// Mitsubishi GX Works2 project: BookEX6_50 Positionning   PLC: Q13UDV

// global labels: Global
VAR_GLOBAL
  bVar0 AT M5000 : BOOL;
  abArray0 AT M5010 : ARRAY [0..49] OF BOOL;
  sStr0 AT D5000 : STRING[199];
  sStr1 AT D5100 : STRING[199];
  sStr2 AT D5200 : STRING[199];
  sStr3 AT D5300 : STRING[199];
  sStr4 AT D5400 : STRING[199];
  sStr5 AT D5500 : STRING[199];
  sStr6 AT D5600 : STRING[199];
  sStr7 AT D5700 : STRING[199];
  sStr8 AT D5800 : STRING[199];
  sStr9 AT D5900 : STRING[199];
  iVar0 AT D4500 : INT;
  iVar1 AT D4501 : INT;
  iVar2 AT D4502 : INT;
  iVar3 AT D4503 : INT;
  iVar4 AT D4504 : INT;
  iVar5 AT D4505 : INT;
  iVar6 AT D4506 : INT;
  iVar7 AT D4507 : INT;
  iVar8 AT D4508 : INT;
  iVar9 AT D4509 : INT;
  dVar0 AT D4510 : DINT;
  dVar1 AT D4512 : DINT;
  dVar2 AT D4514 : DINT;
  dVar3 AT D4516 : DINT;
  dVar4 AT D4518 : DINT;
  dVar5 AT D4520 : DINT;
  dVar6 AT D4522 : DINT;
  dVar7 AT D4524 : DINT;
  dVar8 AT D4526 : DINT;
  dVar9 AT D4528 : DINT;
  wVar0 AT D4530 : WORD;
  wVar1 AT D4531 : WORD;
  wVar2 AT D4532 : WORD;
  wVar3 AT D4533 : WORD;
  wVar4 AT D4534 : WORD;
  wVar5 AT D4535 : WORD;
  wVar6 AT D4536 : WORD;
  wVar7 AT D4537 : WORD;
  wVar8 AT D4538 : WORD;
  wVar9 AT D4539 : WORD;
  dwVar0 AT D4540 : DWORD;
  dwVar1 AT D4542 : DWORD;
  dwVar2 AT D4544 : DWORD;
  dwVar3 AT D4546 : DWORD;
  dwVar4 AT D4548 : DWORD;
  dwVar5 AT D4550 : DWORD;
  dwVar6 AT D4552 : DWORD;
  dwVar7 AT D4554 : DWORD;
  dwVar8 AT D4556 : DWORD;
  dwVar9 AT D4558 : DWORD;
  fsVar0 AT D4560 : REAL;
  fsVar1 AT D4562 : REAL;
  fsVar2 AT D4564 : REAL;
  fsVar3 AT D4566 : REAL;
  fsVar4 AT D4568 : REAL;
  fsVar5 AT D4570 : REAL;
  fsVar6 AT D4572 : REAL;
  fsVar7 AT D4574 : REAL;
  fsVar8 AT D4576 : REAL;
  fsVar9 AT D4578 : REAL;
  fdVar0 AT D4580 : LREAL;
  tTime0 AT D4620 : TIME;
  tTime1 AT D4622 : TIME;
  tTime2 AT D4624 : TIME;
  tTime3 AT D4626 : TIME;
  tTime4 AT D4628 : TIME;
  tTime5 AT D4630 : TIME;
  tTime6 AT D4632 : TIME;
  tTime7 AT D4634 : TIME;
  tTime8 AT D4636 : TIME;
  tTime9 AT D4638 : TIME;
  tTime10 AT D4640 : TIME;
  bVar1 AT M5001 : BOOL;
  bVar2 AT M5002 : BOOL;
  bVar3 AT M5003 : BOOL;
  bVar4 AT M5004 : BOOL;
  bVar5 AT M5005 : BOOL;
  bVar6 AT M5006 : BOOL;
  bVar7 AT M5007 : BOOL;
  bVar8 AT M5008 : BOOL;
  bVar9 AT M5009 : BOOL;
  abArray1 AT M5060 : ARRAY [0..49] OF BOOL;
  abArray2 AT M5110 : ARRAY [0..49] OF BOOL;
  abArray3 AT M5160 : ARRAY [0..49] OF BOOL;
  abArray4 AT M5210 : ARRAY [0..49] OF BOOL;
  abArray5 AT M5260 : ARRAY [0..49] OF BOOL;
  abArray6 AT M5310 : ARRAY [0..49] OF BOOL;
  abArray7 AT M5360 : ARRAY [0..49] OF BOOL;
  abArray8 AT M5410 : ARRAY [0..49] OF BOOL;
  abArray9 AT M5460 : ARRAY [0..49] OF BOOL;
  fdVar1 AT D4584 : LREAL;
  fdVar2 AT D4588 : LREAL;
  fdVar3 AT D4592 : LREAL;
  fdVar4 AT D4596 : LREAL;
  fdVar5 AT D4600 : LREAL;
  fdVar6 AT D4604 : LREAL;
  fdVar7 AT D4608 : LREAL;
  fdVar8 AT D4612 : LREAL;
  fdVar9 AT D4616 : LREAL;
  afsPen0 AT D2000 : ARRAY [0..499] OF REAL;
  afsPen1 AT D3000 : ARRAY [0..499] OF REAL;
END_VAR
// user libraries (not included): HMI

PROGRAM ExPINIT
VAR
  bReqCmd : BOOL;
  bExeFlag : BOOL;
  bMemFlag : BOOL;
  aCtrlData : ARRAY [0..1] OF INT;
  abComp : ARRAY [0..1] OF BOOL;
  iErrCode : INT;
END_VAR
(* structured ladder/FBD written out as ST: instructions are called as NAME(EN, inputs, outputs); _pN, _eN, _tN stand for wires *)
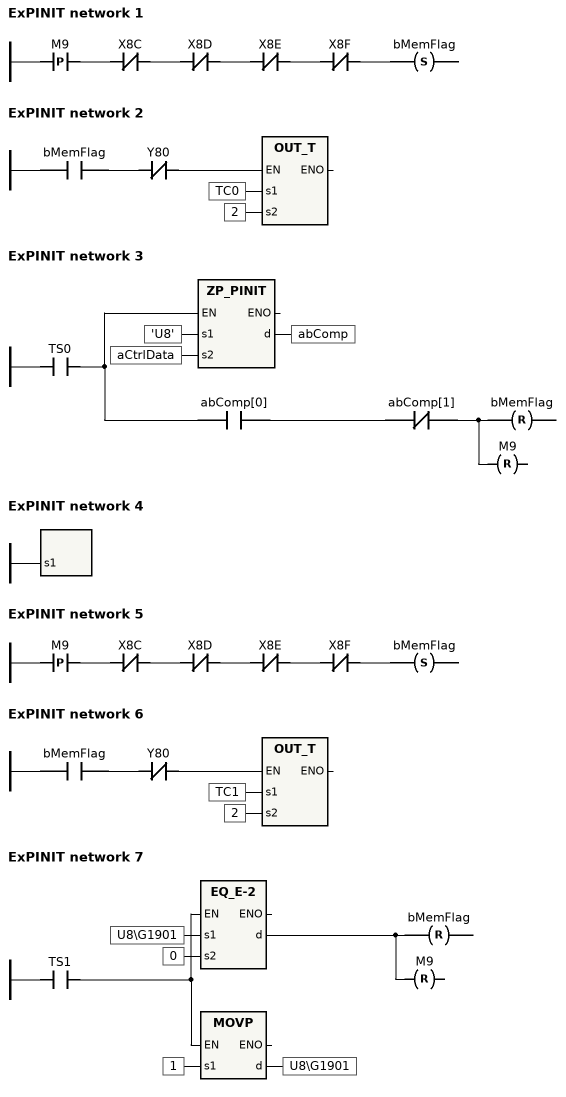
(* network 1 *)
SET(LDP(TRUE, M9) AND NOT X8C AND NOT X8D AND NOT X8E AND NOT X8F, bMemFlag);
(* network 2 *)
OUT_T(bMemFlag AND NOT Y80, TC0, 2);
(* network 3 *)
ZP_PINIT(TS0, 'U8', aCtrlData, abComp);
_p1 := TS0 AND abComp[0] AND NOT abComp[1];
RST(_p1, bMemFlag);
RST(_p1, M9);
(* network 4 *)
(* element kind 10  <- TRUE *)
(* network 5 *)
SET(LDP(TRUE, M9) AND NOT X8C AND NOT X8D AND NOT X8E AND NOT X8F, bMemFlag);
(* network 6 *)
OUT_T(bMemFlag AND NOT Y80, TC1, 2);
(* network 7 *)
MOVP(TS1, 1, U8\G1901);
EQ_E(TS1, U8\G1901, 0, _t1);
RST(_t1, bMemFlag);
RST(_t1, M9);
END_PROGRAM

PROGRAM ExABRST
VAR
  bReqCmd : BOOL;
  bExeFlag : BOOL;
  bMemFlag : BOOL;
  aCtrlData : ARRAY [0..7] OF INT;
  abComp : ARRAY [0..1] OF BOOL;
  iErrCode : INT;
END_VAR
(* structured ladder/FBD written out as ST: instructions are called as NAME(EN, inputs, outputs); _pN, _eN, _tN stand for wires *)
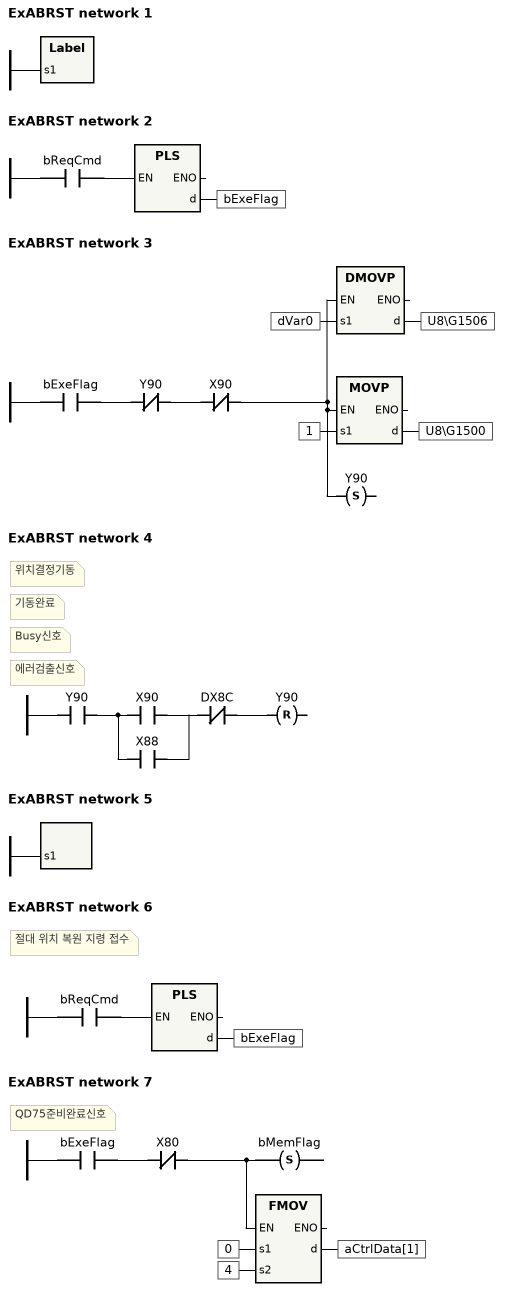
(* network 1 *)
(* element kind 9 Label <- TRUE *)
(* network 2 *)
PLS(bReqCmd, bExeFlag);
(* network 3 *)
_p1 := bExeFlag AND NOT Y90 AND NOT X90;
DMOVP(_p1, dVar0, U8\G1506);
MOVP(_p1, 1, U8\G1500);
SET(_p1, Y90);
(* network 4 *)
(* 위치결정기동 *)
(* 기동완료 *)
(* Busy신호 *)
(* 에러검출신호 *)
RST(((Y90 AND X90) OR (Y90 AND X88)) AND NOT DX8C, Y90);
(* network 5 *)
(* element kind 10  <- TRUE *)
(* network 6 Label: *)
(* 절대 위치 복원 지령 접수 *)
PLS(bReqCmd, bExeFlag);
(* network 7 *)
(* QD75준비완료신호 *)
_p1 := bExeFlag AND NOT X80;
SET(_p1, bMemFlag);
FMOV(_p1, 0, 4, aCtrlData[1]);
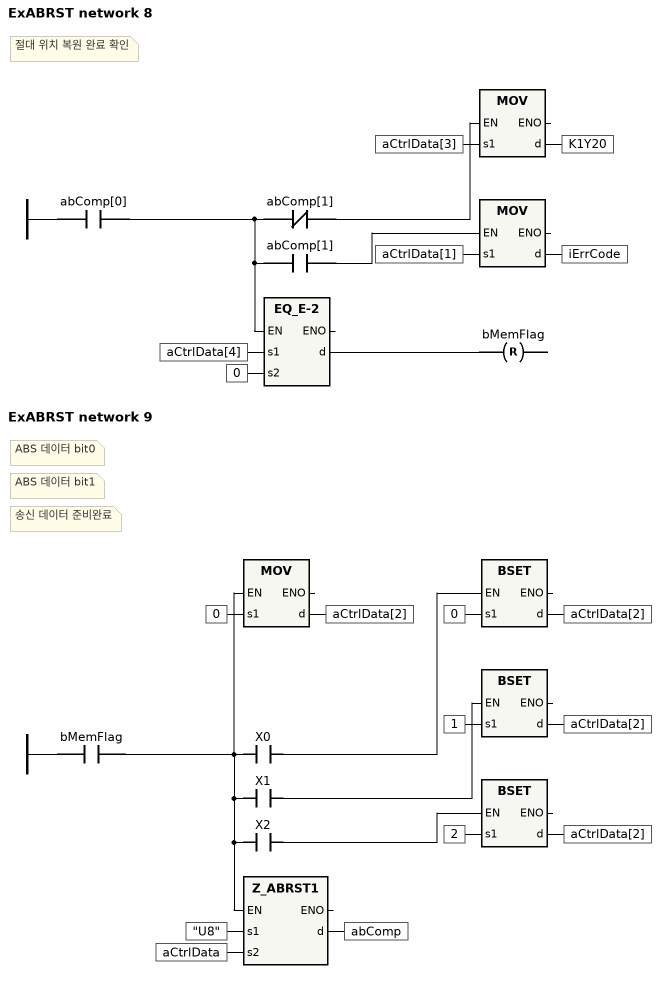
(* network 8 *)
(* 절대 위치 복원 완료 확인 *)
MOV(abComp[0] AND NOT abComp[1], aCtrlData[3], K1Y20);
MOV(abComp[0] AND abComp[1], aCtrlData[1], iErrCode);
EQ_E(abComp[0], aCtrlData[4], 0, _t1);
RST(_t1, bMemFlag);
(* network 9 *)
(* ABS 데이터 bit0 *)
(* ABS 데이터 bit1 *)
(* 송신 데이터 준비완료 *)
MOV(bMemFlag, 0, aCtrlData[2]);
BSET(bMemFlag AND X0, 0, aCtrlData[2]);
BSET(bMemFlag AND X1, 1, aCtrlData[2]);
BSET(bMemFlag AND X2, 2, aCtrlData[2]);
Z_ABRST1(bMemFlag, "U8", aCtrlData, abComp);
END_PROGRAM

PROGRAM ExPSTRT
VAR
  bReqCmd : BOOL;
  bExeFlag : BOOL;
  bMemFlag : BOOL;
  aCtrlData : ARRAY [0..2] OF INT;
  abComp : ARRAY [0..1] OF BOOL;
  iErrCode : INT;
END_VAR
(* structured ladder/FBD written out as ST: instructions are called as NAME(EN, inputs, outputs); _pN, _eN, _tN stand for wires *)
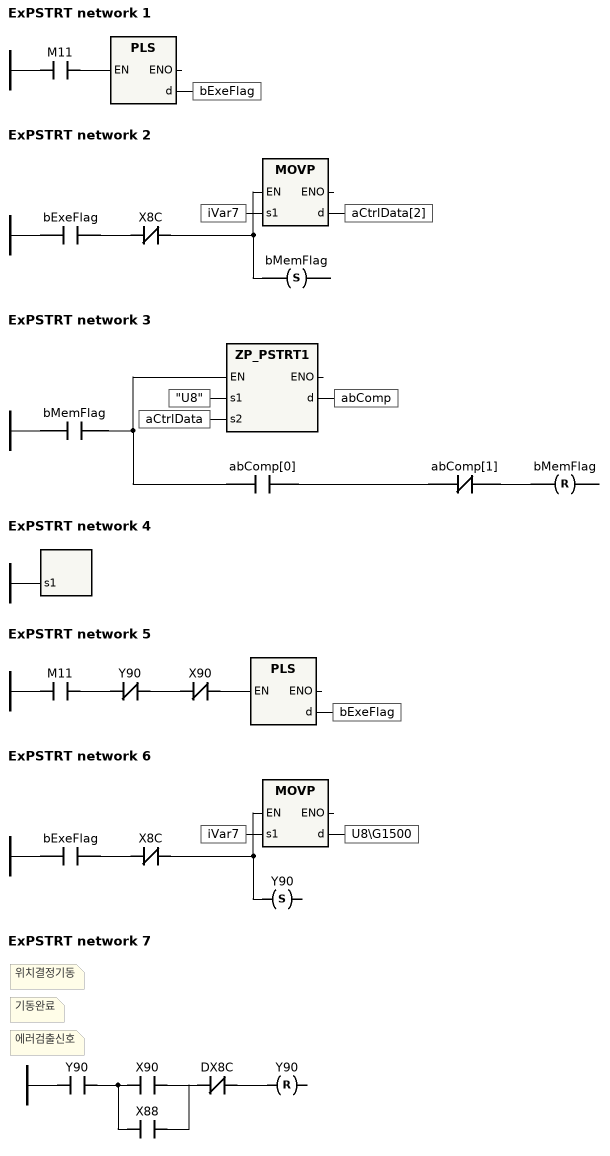
(* network 1 *)
PLS(M11, bExeFlag);
(* network 2 *)
_p1 := bExeFlag AND NOT X8C;
MOVP(_p1, iVar7, aCtrlData[2]);
SET(_p1, bMemFlag);
(* network 3 *)
ZP_PSTRT1(bMemFlag, "U8", aCtrlData, abComp);
RST(bMemFlag AND abComp[0] AND NOT abComp[1], bMemFlag);
(* network 4 *)
(* element kind 10  <- TRUE *)
(* network 5 Label: *)
PLS(M11 AND NOT Y90 AND NOT X90, bExeFlag);
(* network 6 *)
_p1 := bExeFlag AND NOT X8C;
MOVP(_p1, iVar7, U8\G1500);
SET(_p1, Y90);
(* network 7 *)
(* 위치결정기동 *)
(* 기동완료 *)
(* 에러검출신호 *)
RST(((Y90 AND X90) OR (Y90 AND X88)) AND NOT DX8C, Y90);
END_PROGRAM

PROGRAM ExTEACH
VAR
  bReqCmd : BOOL;
  bExeFlag : BOOL;
  bMemFlag : BOOL;
  aCtrlData : ARRAY [0..3] OF INT;
  abComp : ARRAY [0..1] OF BOOL;
  iErrCode : INT;
END_VAR
(* structured ladder/FBD written out as ST: instructions are called as NAME(EN, inputs, outputs); _pN, _eN, _tN stand for wires *)
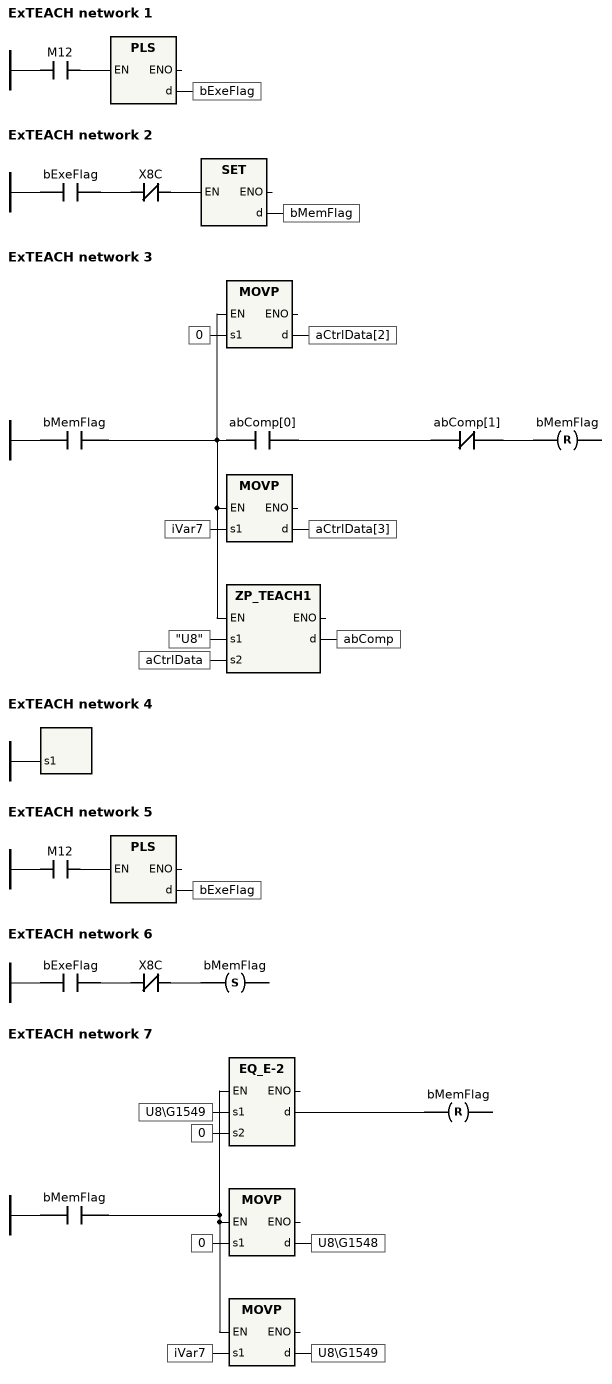
(* network 1 *)
PLS(M12, bExeFlag);
(* network 2 *)
SET(bExeFlag AND NOT X8C, bMemFlag);
(* network 3 *)
MOVP(bMemFlag, 0, aCtrlData[2]);
MOVP(bMemFlag, iVar7, aCtrlData[3]);
ZP_TEACH1(bMemFlag, "U8", aCtrlData, abComp);
RST(bMemFlag AND abComp[0] AND NOT abComp[1], bMemFlag);
(* network 4 *)
(* element kind 10  <- TRUE *)
(* network 5 *)
PLS(M12, bExeFlag);
(* network 6 *)
SET(bExeFlag AND NOT X8C, bMemFlag);
(* network 7 *)
MOVP(bMemFlag, 0, U8\G1548);
MOVP(bMemFlag, iVar7, U8\G1549);
EQ_E(bMemFlag, U8\G1549, 0, _t1);
RST(_t1, bMemFlag);
END_PROGRAM

PROGRAM ExPFWRT
VAR
  bReqCmd : BOOL;
  bExeFlag : BOOL;
  bMemFlag : BOOL;
  aCtrlData : ARRAY [0..1] OF INT;
  abComp : ARRAY [0..1] OF BOOL;
  iErrCode : INT;
END_VAR
(* structured ladder/FBD written out as ST: instructions are called as NAME(EN, inputs, outputs); _pN, _eN, _tN stand for wires *)
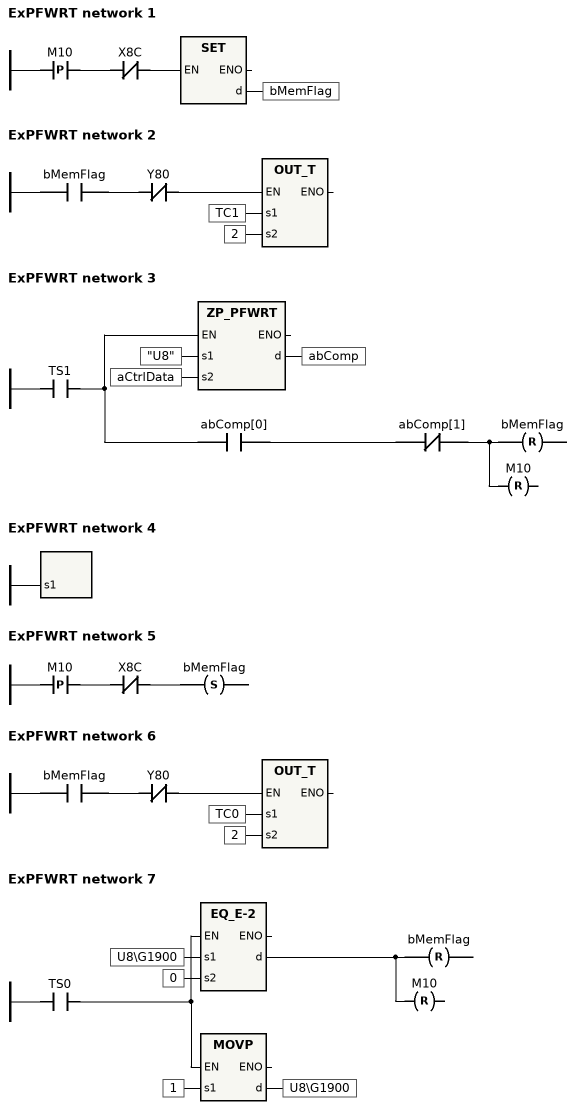
(* network 1 *)
SET(LDP(TRUE, M10) AND NOT X8C, bMemFlag);
(* network 2 *)
OUT_T(bMemFlag AND NOT Y80, TC1, 2);
(* network 3 *)
ZP_PFWRT(TS1, "U8", aCtrlData, abComp);
_p1 := TS1 AND abComp[0] AND NOT abComp[1];
RST(_p1, bMemFlag);
RST(_p1, M10);
(* network 4 *)
(* element kind 10  <- TRUE *)
(* network 5 *)
SET(LDP(TRUE, M10) AND NOT X8C, bMemFlag);
(* network 6 *)
OUT_T(bMemFlag AND NOT Y80, TC0, 2);
(* network 7 *)
MOVP(TS0, 1, U8\G1900);
EQ_E(TS0, U8\G1900, 0, _t1);
RST(_t1, bMemFlag);
RST(_t1, M10);
END_PROGRAM

FUNCTION_BLOCK ms2Ready
VAR_INPUT
  b_EN : BOOL;
  i_Start_IO_No : INT;  (* Module XY addr *)
END_VAR
VAR_OUTPUT
  b_ENO : BOOL;
  b_Ready : BOOL;
END_VAR
VAR
  bRdy77 : BOOL;
  bRdyCPU : BOOL;
END_VAR
VAR_OUTPUT
  b_AllAxis : BOOL;
  b_OK : BOOL;
END_VAR
VAR
  bSync77 : BOOL;
  bReady : BOOL;
  bAllAxis : BOOL;
END_VAR
;
b_ENO := b_EN;
Z0 := i_Start_IO_No * 16;
bRdy77 := X0Z0;
bSync77 := X1Z0;
bRdyCPU := Y0Z0;

IF NOT b_EN  THEN
	bReady := FALSE;
	bAllAxis := FALSE;
	b_OK := FALSE;
ELSE
	bReady := NOT SM0;
	bAllAxis := bRdyCPU AND bSync77;
	b_OK := bRdyCPU AND bRdy77 AND bSync77;
END_IF;

b_Ready := bReady;
b_AllAxis := bAllAxis;
END_FUNCTION_BLOCK

FUNCTION_BLOCK ms2Status
VAR_INPUT
  b_EN : BOOL;
  i_Start_IO_No : INT;  (* Module XY addr *)
  i_Axis : INT;  (* Axis No *)
END_VAR
VAR_OUTPUT
  b_ENO : BOOL;
  i_Status : INT;
  i_Error : INT;
END_VAR
VAR
  bRes : BOOL;
  AxisOff : INT;
  iTmp : INT;
END_VAR
VAR_OUTPUT
  d_CurrVal : DINT;
END_VAR
VAR
  dTmp : DINT;
END_VAR
VAR_OUTPUT
  d_CurrSpd : DINT;
  i_Warn : INT;
  d_TargVal : DINT;
  d_TargSpd : DINT;
  d_MacVal : DINT;
  w_Flag : WORD;
  w_Signal : WORD;
END_VAR
;
b_ENO := b_EN;
IF NOT LDP(TRUE, b_EN) THEN
	RETURN;
END_IF;
AxisOff := (i_Axis - 1) * 100;
bRes := FROM( TRUE, i_Start_IO_No, AxisOff+809, 1, iTmp);
i_Status := iTmp;
bRes := FROM( TRUE, i_Start_IO_No, AxisOff+806, 1, iTmp);
i_Error := iTmp;
bRes := FROM( TRUE, i_Start_IO_No, AxisOff+807, 1, iTmp);
i_Warn := iTmp;
bRes := DFRO( TRUE, i_Start_IO_No, AxisOff+800, 1, dTmp);
d_CurrVal := dTmp;
bRes := DFRO( TRUE, i_Start_IO_No, AxisOff+802, 1, dTmp);
d_MacVal := dTmp;
bRes := DFRO( TRUE, i_Start_IO_No, AxisOff+810, 1, dTmp);
d_CurrSpd := dTmp;
bRes := DFRO( TRUE, i_Start_IO_No, AxisOff+818, 1, dTmp);
d_TargVal := dTmp;
bRes := DFRO( TRUE, i_Start_IO_No, AxisOff+820, 1, dTmp);
d_TargSpd := dTmp;
bRes := FROM( TRUE, i_Start_IO_No, AxisOff+817, 1, iTmp);
w_Flag := INT_TO_WORD(iTmp);
bRes := FROM( TRUE, i_Start_IO_No, AxisOff+816, 1, iTmp);
w_Signal := INT_TO_WORD(iTmp);

(* 축 동작상태
		-2：스텝 대기중
		-1：에러 발생중
		0：대기중
		1：정지중
		2：보간중
		3：JOG 운전중
		4：수동 펄서 운전중
		5：해석중
		6：특수 기동 대기중
		7：원점복귀중
		8：위치제어중
		9：속도제어중
		10：속도·위치제어의 속도제어중
		11：속도·위치제어의 위치제어중
		12：위치·속도제어의 위치제어중
		13：위치·속도제어의 속도제어중
		15：동기제어중
		20：서보 미접속/서보앰프 전원 OFF
		21：서보 OFF 중
		30：제어모드 전환중
		31：속도 제어 모드중
		32：토크 제어 모드중
		33：스톱퍼 제어 모드중
*)
END_FUNCTION_BLOCK

FUNCTION_BLOCK ms2JOG
VAR_INPUT
  b_EN : BOOL;
  i_Start_IO_No : INT;  (* Module XY addr *)
  i_Axis : INT;  (* Axis No *)
  b_CW : BOOL;
  b_CCW : BOOL;
  d_JOGSpd : DINT;
END_VAR
VAR_OUTPUT
  b_ENO : BOOL;
END_VAR
VAR
  bRes : BOOL;
  AxisOff : INT;
  bError : BOOL;
  bBusy : BOOL;
  bReady : BOOL;
  bCW : BOOL;
  bCCW : BOOL;
END_VAR
VAR_INPUT
  b_SetSp : BOOL;
END_VAR
VAR
  bRun : BOOL;
  iCmd : INT;
END_VAR
;
b_ENO := b_EN;
Z0 := i_Start_IO_No * 16;
Z1 := Z0 + i_Axis - 1;
AxisOff := (i_Axis - 1) * 100;
bReady := X0Z0;
bError := X8Z1;
bBusy := XCZ0;

IF LDP(TRUE, b_SetSp) THEN
	bRes	:= TO( TRUE, 0, i_Start_IO_No, AxisOff+1517, 1);
	bRes	:= DTO( TRUE, d_JOGSpd * 10000, i_Start_IO_No, AxisOff+1518, 1);
END_IF;
iCmd := BOOL_TO_INT(b_CW) + BOOL_TO_INT(b_CCW) * 2;
CASE iCmd OF
	0, 3 : 	bCW := FALSE;
				bCCW := FALSE;
	1 : (* CW *)
				bCW := 	bReady AND NOT bError;
	2 : (* CCW *)
				bCCW := 	bReady AND NOT bError;
END_CASE;			 

Y8Z0 :=	bCCW;
Y9Z0 := bCW;
END_FUNCTION_BLOCK

PROGRAM ExJOG
VAR
  RunJog : BOOL;
  ServoRdy : BOOL;
  ReqHOFF : BOOL;
  MemHOFF : BOOL;
  wTmp : WORD;
  CmdHOFF : BOOL;
  ReqHPR : BOOL;
  ReqStop : BOOL;
END_VAR
(* structured ladder/FBD written out as ST: instructions are called as NAME(EN, inputs, outputs); _pN, _eN, _tN stand for wires *)
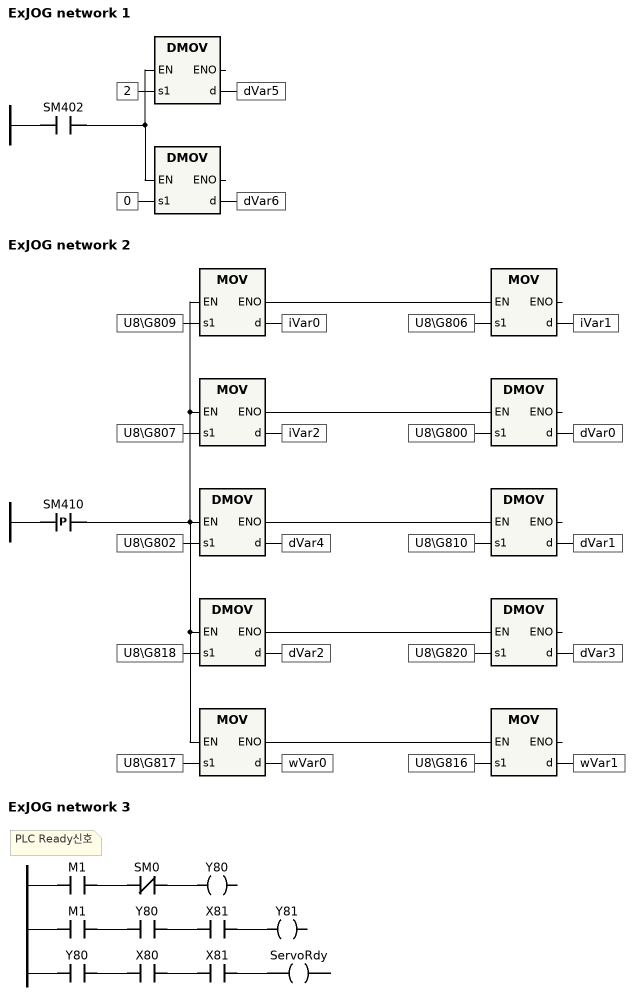
(* network 1 *)
DMOV(SM402, 2, dVar5);
DMOV(SM402, 0, dVar6);
(* network 2 *)
_p1 := LDP(TRUE, SM410);
_e2 := MOV(_p1, U8\G809, iVar0);
MOV(_e2, U8\G806, iVar1);
_e3 := MOV(_p1, U8\G807, iVar2);
DMOV(_e3, U8\G800, dVar0);
_e4 := DMOV(_p1, U8\G802, dVar4);
DMOV(_e4, U8\G810, dVar1);
_e5 := DMOV(_p1, U8\G818, dVar2);
DMOV(_e5, U8\G820, dVar3);
_e6 := MOV(_p1, U8\G817, wVar0);
MOV(_e6, U8\G816, wVar1);
(* network 3 *)
(* PLC Ready신호 *)
Y80 := M1 AND NOT SM0;
Y81 := M1 AND Y80 AND X81;
ServoRdy := Y80 AND X80 AND X81;
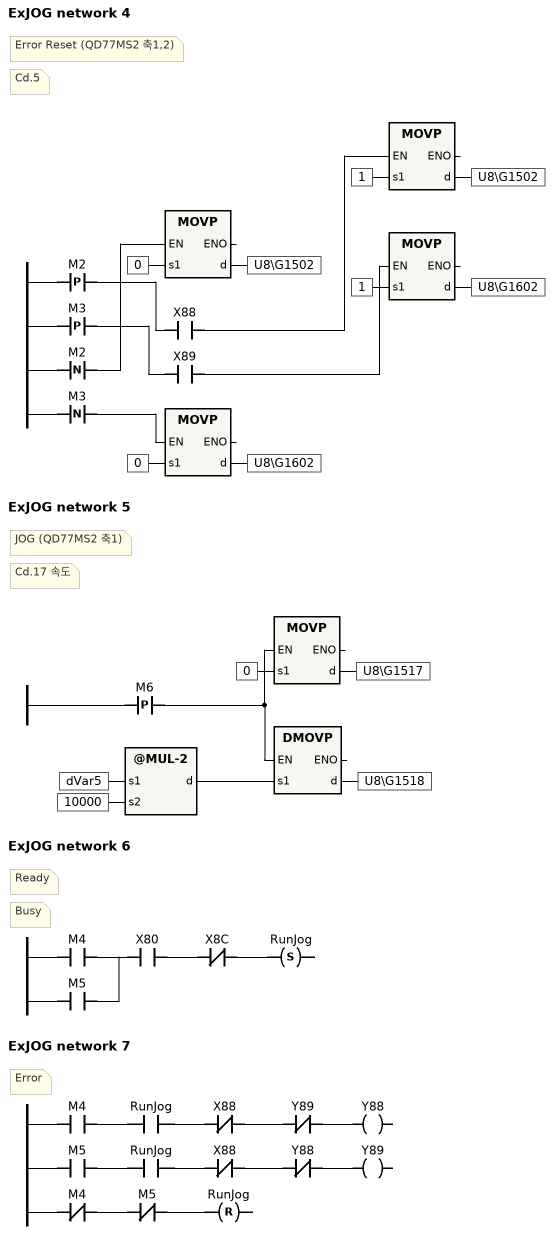
(* network 4 *)
(* Error Reset (QD77MS2 축1,2) *)
(* Cd.5 *)
MOVP(LDP(TRUE, M2) AND X88, 1, U8\G1502);
MOVP(LDP(TRUE, M3) AND X89, 1, U8\G1602);
MOVP(LDF(TRUE, M2), 0, U8\G1502);
MOVP(LDF(TRUE, M3), 0, U8\G1602);
(* network 5 *)
(* JOG (QD77MS2 축1) *)
(* Cd.17 속도 *)
_p1 := LDP(TRUE, M6);
MOVP(_p1, 0, U8\G1517);
DMOVP(_p1, @MUL-2(dVar5, 10000), U8\G1518);
(* network 6 *)
(* Ready *)
(* Busy *)
SET(((M4 OR M5) AND X80) AND NOT X8C, RunJog);
(* network 7 *)
(* Error *)
Y88 := M4 AND RunJog AND NOT X88 AND NOT Y89;
Y89 := M5 AND RunJog AND NOT X88 AND NOT Y88;
RST(NOT M4 AND NOT M5, RunJog);
END_PROGRAM

PROGRAM ExDataSet
VAR
  RunJog : BOOL;
  ServoRdy : BOOL;
  ReqHOFF : BOOL;
  MemHOFF : BOOL;
  wTmp : WORD;
  CmdHOFF : BOOL;
  ReqHPR : BOOL;
  ReqStop : BOOL;
END_VAR
(* structured ladder/FBD written out as ST: instructions are called as NAME(EN, inputs, outputs); _pN, _eN, _tN stand for wires *)
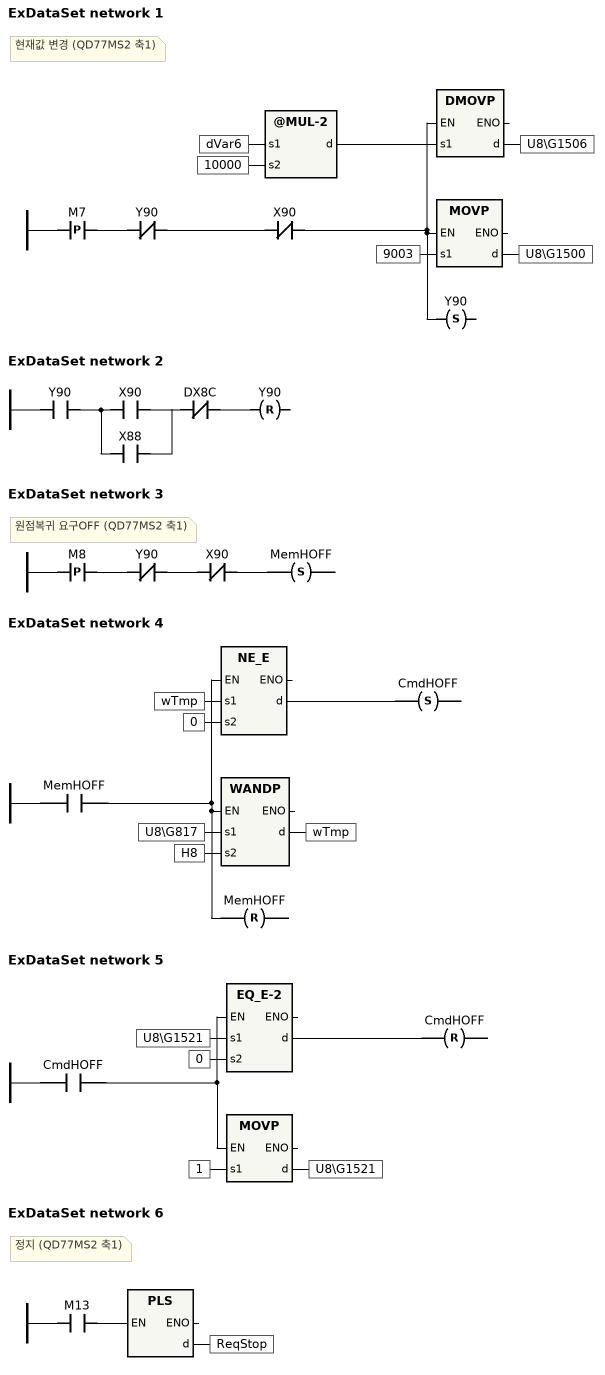
(* network 1 *)
(* 현재값 변경 (QD77MS2 축1) *)
_p1 := LDP(TRUE, M7) AND NOT Y90 AND NOT X90;
DMOVP(_p1, @MUL-2(dVar6, 10000), U8\G1506);
MOVP(_p1, 9003, U8\G1500);
SET(_p1, Y90);
(* network 2 *)
RST(((Y90 AND X90) OR (Y90 AND X88)) AND NOT DX8C, Y90);
(* network 3 *)
(* 원점복귀 요구OFF (QD77MS2 축1) *)
SET(LDP(TRUE, M8) AND NOT Y90 AND NOT X90, MemHOFF);
(* network 4 *)
WANDP(MemHOFF, U8\G817, H8, wTmp);
NE_E(MemHOFF, wTmp, 0, _t1);
SET(_t1, CmdHOFF);
RST(MemHOFF, MemHOFF);
(* network 5 *)
MOVP(CmdHOFF, 1, U8\G1521);
EQ_E(CmdHOFF, U8\G1521, 0, _t1);
RST(_t1, CmdHOFF);
(* network 6 *)
(* 정지 (QD77MS2 축1) *)
PLS(M13, ReqStop);
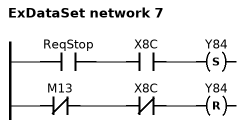
(* network 7 *)
SET(ReqStop AND X8C, Y84);
RST(NOT M13 AND NOT X8C, Y84);
END_PROGRAM

PROGRAM ExPSTRT2
VAR
  bReqCmd : BOOL;
  bExeFlag : BOOL;
  bMemFlag : BOOL;
  aCtrlData : ARRAY [0..2] OF INT;
  abComp : ARRAY [0..1] OF BOOL;
  iErrCode : INT;
  Buffer : ARRAY [0..4] OF DINT;
END_VAR
(* structured ladder/FBD written out as ST: instructions are called as NAME(EN, inputs, outputs); _pN, _eN, _tN stand for wires *)
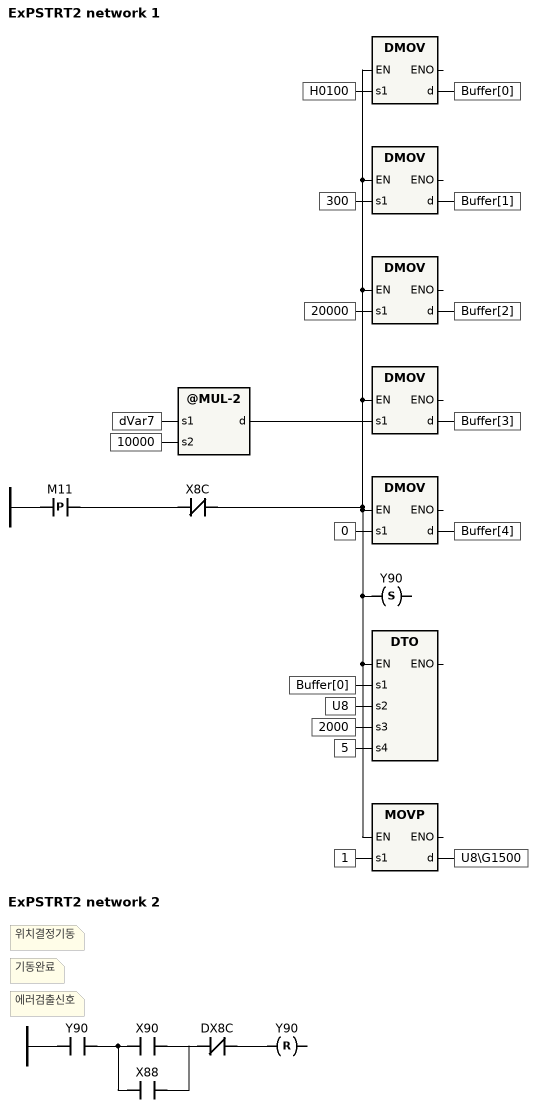
(* network 1 *)
_p1 := LDP(TRUE, M11) AND NOT X8C;
DMOV(_p1, H0100, Buffer[0]);
DMOV(_p1, 300, Buffer[1]);
DMOV(_p1, 20000, Buffer[2]);
DMOV(_p1, @MUL-2(dVar7, 10000), Buffer[3]);
DMOV(_p1, 0, Buffer[4]);
DTO(_p1, Buffer[0], U8, 2000, 5);
MOVP(_p1, 1, U8\G1500);
SET(_p1, Y90);
(* network 2 *)
(* 위치결정기동 *)
(* 기동완료 *)
(* 에러검출신호 *)
RST(((Y90 AND X90) OR (Y90 AND X88)) AND NOT DX8C, Y90);
END_PROGRAM

PROGRAM ExJOG_ST
VAR
  RunJog : BOOL;
  ServoRdy : BOOL;
  ReqHOFF : BOOL;
  MemHOFF : BOOL;
  wTmp : WORD;
  CmdHOFF : BOOL;
  ReqHPR : BOOL;
  ReqStop : BOOL;
  ms2Status_1 : ms2Status;
  ms2Ready_1 : ms2Ready;
  ms2Reset_1 : ms2Reset;
  ms2JOG_1 : ms2JOG;
  ms2Stop_1 : ms2Stop;
  ms2HPR_1 : ms2HPR;
  ms2PosRun_1 : ms2PosRun;
  ms2Run_1 : ms2Run;
END_VAR
(* structured ladder/FBD written out as ST: instructions are called as NAME(EN, inputs, outputs); _pN, _eN, _tN stand for wires *)
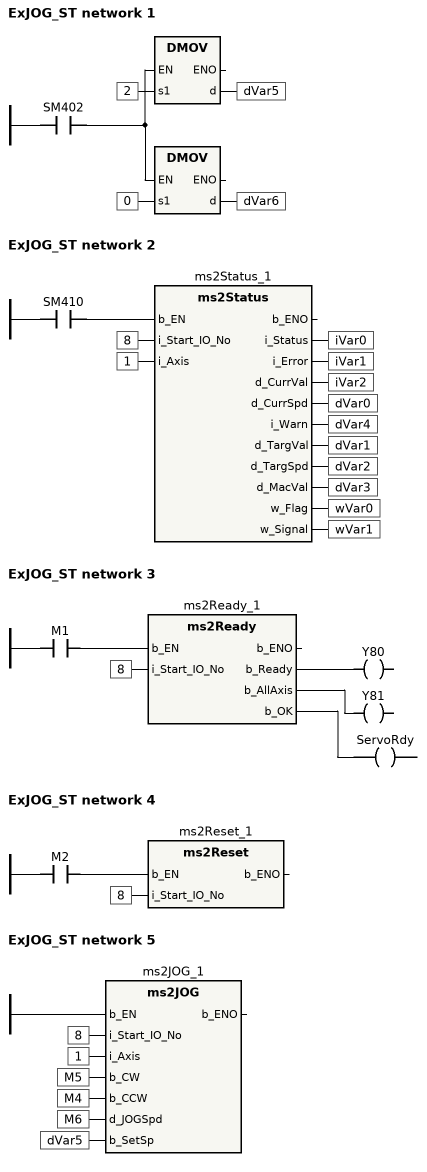
(* network 1 *)
DMOV(SM402, 2, dVar5);
DMOV(SM402, 0, dVar6);
(* network 2 *)
ms2Status_1(b_EN := SM410, i_Start_IO_No := 8, i_Axis := 1, i_Status => iVar0, i_Error => iVar1, d_CurrVal => iVar2, d_CurrSpd => dVar0, i_Warn => dVar4, d_TargVal => dVar1, d_TargSpd => dVar2, d_MacVal => dVar3, w_Flag => wVar0, w_Signal => wVar1);
(* network 3 *)
ms2Ready_1(b_EN := M1, i_Start_IO_No := 8);
Y80 := ms2Ready_1.b_Ready;
Y81 := ms2Ready_1.b_AllAxis;
ServoRdy := ms2Ready_1.b_OK;
(* network 4 *)
ms2Reset_1(b_EN := M2, i_Start_IO_No := 8);
(* network 5 *)
ms2JOG_1(b_EN := TRUE, i_Start_IO_No := 8, i_Axis := 1, b_CW := M5, b_CCW := M4, d_JOGSpd := M6, b_SetSp := dVar5);
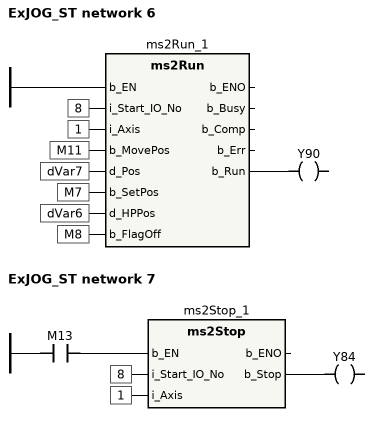
(* network 6 *)
ms2Run_1(b_EN := TRUE, i_Start_IO_No := 8, i_Axis := 1, b_MovePos := M11, d_Pos := dVar7, b_SetPos := M7, d_HPPos := dVar6, b_FlagOff := M8);
Y90 := ms2Run_1.b_Run;
(* network 7 *)
ms2Stop_1(b_EN := M13, i_Start_IO_No := 8, i_Axis := 1);
Y84 := ms2Stop_1.b_Stop;
END_PROGRAM

FUNCTION_BLOCK ms2Reset
VAR_INPUT
  b_EN : BOOL;
  i_Start_IO_No : INT;
END_VAR
VAR_OUTPUT
  b_ENO : BOOL;
END_VAR
VAR
  Result : BOOL;
  bError1 : BOOL;
  bError2 : BOOL;
  iCmd : INT;
END_VAR
(* 사용중인 축에 에러가 있으면 reset한다. *)
b_ENO 			:= b_EN;
Z0 := i_Start_IO_No * 16;
bError1 := X8Z0;
bError2 := X9Z0;

IF LDF(TRUE, b_EN) THEN
	iCmd := 0;
	Result := TO( TRUE,  iCmd,  i_Start_IO_No, 1502, 1);
	Result := TO( TRUE,  iCmd, i_Start_IO_No, 1602, 1);
END_IF;
IF NOT b_EN THEN
		RETURN;
END_IF;
IF LDP(TRUE, b_EN) THEN
	iCmd := 1;
	IF bError1 THEN Result := TO( TRUE, iCmd, i_Start_IO_No, 1502, 1); END_IF;
	IF bError1 THEN Result := TO( TRUE, iCmd, i_Start_IO_No, 1602, 1); END_IF;
 END_IF;
END_FUNCTION_BLOCK

FUNCTION_BLOCK ms2PosRun
VAR_INPUT
  b_EN : BOOL;
END_VAR
VAR_OUTPUT
  b_ENO : BOOL;
END_VAR
VAR
  AxisOff : INT;
END_VAR
VAR_INPUT
  i_Start_IO_No : INT;
  i_Axis : INT;
  b_MovePos : BOOL;
END_VAR
VAR
  abComp : ARRAY [0..1] OF BOOL;
  SeqNo : INT;
  Buffer : ARRAY [0..4] OF DINT;
END_VAR
VAR_OUTPUT
  b_Busy : BOOL;
  b_Comp : BOOL;
  b_Err : BOOL;
END_VAR
VAR_INPUT
  d_Pos : DINT;
END_VAR
VAR
  Result : BOOL;
END_VAR
;
b_ENO 			:= b_EN;
Z0 := i_Start_IO_No * 16;
Z1 := Z0 + i_Axis - 1;
AxisOff 		:= (i_Axis -1) * 100;

CASE SeqNo OF 
	0 :	(* Wait *)
				IF LDP(TRUE, b_MovePos) AND NOT XCZ1 THEN 
						SeqNo := 1;								
				END_IF;
	1 :	(* Run *)	
				Buffer[0] := H0100;
				Buffer[1] := 300;
				Buffer[2] := 20000;
				Buffer[3] := d_Pos * 10000;
				Buffer[4] := 0;
				Result := DTO( TRUE, Buffer[0], i_Start_IO_No, 2000 + AxisOff * 6000, 5);
				Result := TO( TRUE, 1, i_Start_IO_No, 1500 + AxisOff, 1);
				Y10Z1 := TRUE;
				SeqNo := 2;
	2 :	(* Wait complete *)	
				IF Y10Z1 AND NOT XCZ1 AND (X10Z1 OR X8Z1) THEN
						Y10Z1 := FALSE;
						SeqNo := 3;
				END_IF;
				b_Busy := XCZ1;
				b_Comp := X10Z1;
				b_Err := X8Z1;
	3 : (* Stop *)
				IF NOT Y10Z1 THEN
						SeqNo := 0;
				END_IF;
END_CASE;
END_FUNCTION_BLOCK

FUNCTION_BLOCK ms2HPR
VAR_INPUT
  b_EN : BOOL;
  b_SetPos : BOOL;
  d_HPPos : DINT;
END_VAR
VAR_OUTPUT
  b_ENO : BOOL;
END_VAR
VAR
  AxisOff : INT;
  SlotNo : INT;
  dData : DINT;
  bRun : BOOL;
  Result : BOOL;
  wTmp : WORD;
END_VAR
VAR_INPUT
  i_Start_IO_No : INT;
  b_FlagOff : BOOL;
  i_Axis : INT;
END_VAR
;
b_ENO 			:= b_EN;
Z0 := i_Start_IO_No * 16;
Z1 := Z0 + i_Axis - 1;
AxisOff 		:= (i_Axis -1) * 100;

IF LDP(TRUE, b_SetPos) AND NOT Y10Z1 AND NOT X10Z1 THEN
		dData := d_HPPos * 10000;
		Result := DTO( TRUE, dData, i_Start_IO_No, 1506 + AxisOff, 1);
		Result := TO( TRUE, 9003, i_Start_IO_No, 1500 + AxisOff, 1);
		Y10Z1 := TRUE;
END_IF;
IF b_SetPos AND Y10Z1 AND NOT XCZ1 AND (X10Z1 OR X8Z1) THEN
		Y10Z1 := FALSE;
END_IF;

IF LDP(TRUE, b_FlagOff) AND NOT Y10Z1 AND NOT X10Z1 THEN
		Result := FROM( TRUE, i_Start_IO_No, 817 + AxisOff, 1, wTmp);
		IF (wTmp AND H0008) <> 0 THEN
				Result := TO( TRUE, 1, i_Start_IO_No, 1521 + AxisOff, 1);
		END_IF;
END_IF;
END_FUNCTION_BLOCK

FUNCTION_BLOCK ms2Stop
VAR_INPUT
  b_EN : BOOL;
  i_Start_IO_No : INT;
END_VAR
VAR_OUTPUT
  b_ENO : BOOL;
END_VAR
VAR
  bStop : BOOL;
END_VAR
VAR_INPUT
  i_Axis : INT;  (* Axis No *)
END_VAR
VAR_OUTPUT
  b_Stop : BOOL;
END_VAR
; 
b_ENO 			:= b_EN;
Z0 := i_Start_IO_No * 16;
Z1 := Z0 + i_Axis - 1;
IF LDP(TRUE, b_EN) AND XCZ1 THEN bStop := TRUE; END_IF;
IF NOT b_EN AND NOT XCZ1 THEN bStop := FALSE; END_IF;

b_Stop := bStop;
END_FUNCTION_BLOCK

FUNCTION_BLOCK ms2Run
VAR_INPUT
  b_EN : BOOL;
END_VAR
VAR_OUTPUT
  b_ENO : BOOL;
END_VAR
VAR
  AxisOff : INT;
END_VAR
VAR_INPUT
  i_Start_IO_No : INT;
  i_Axis : INT;
  b_MovePos : BOOL;
END_VAR
VAR
  SeqNo : INT;
  Buffer : ARRAY [0..4] OF DINT;
END_VAR
VAR_OUTPUT
  b_Busy : BOOL;
  b_Comp : BOOL;
  b_Err : BOOL;
END_VAR
VAR_INPUT
  d_Pos : DINT;
END_VAR
VAR
  Result : BOOL;
END_VAR
VAR_INPUT
  b_SetPos : BOOL;
  d_HPPos : DINT;
  b_FlagOff : BOOL;
END_VAR
VAR
  wTmp : WORD;
END_VAR
VAR_OUTPUT
  b_Run : BOOL;
END_VAR
VAR
  bRunOut : BOOL;
END_VAR
;
b_ENO 			:= b_EN;
Z0 := i_Start_IO_No * 16;
Z1 := Z0 + i_Axis - 1;
AxisOff 		:= (i_Axis -1) * 100;

CASE SeqNo OF 
	0 :	(* Wait *)
				IF LDP(TRUE, b_MovePos) AND NOT XCZ1 THEN 
						SeqNo := 1;								
				END_IF;
				IF LDP(TRUE, b_SetPos) AND NOT Y10Z1 AND NOT X10Z1 THEN 
						SeqNo := 10;								
				END_IF;
				IF LDP(TRUE, b_FlagOff) AND NOT Y10Z1 AND NOT X10Z1 THEN 
						SeqNo := 20;								
				END_IF;
	1 :	(* Run *)	
				Buffer[0] := H0100;
				Buffer[1] := 300;
				Buffer[2] := 20000;
				Buffer[3] := d_Pos * 10000;
				Buffer[4] := 0;
				Result := DTO( TRUE, Buffer[0], i_Start_IO_No, 2000 + AxisOff * 6000, 5);
				Result := TO( TRUE, 1, i_Start_IO_No, 1500 + AxisOff, 1);
				bRunOut := TRUE;
				SeqNo := 2;
	2 :	(* Wait complete *)	
				IF Y10Z1 AND NOT XCZ1 AND (X10Z1 OR X8Z1) THEN
						bRunOut := FALSE;
						SeqNo := 3;
				END_IF;
				b_Busy := XCZ1;
				b_Comp := X10Z1;
				b_Err := X8Z1;
	3 : (* Stop *)
				IF NOT Y10Z1 THEN
						SeqNo := 0;
				END_IF;
	10 : (* Set Current Position *)
				Buffer[0] := d_HPPos * 10000;
				Result := DTO( TRUE, Buffer[0], i_Start_IO_No, 1506 + AxisOff, 1);
				Result := TO( TRUE, 9003, i_Start_IO_No, 1500 + AxisOff, 1);
				bRunOut := TRUE;
				SeqNo := 11;
	11 : (* Wait *)
				IF b_SetPos AND Y10Z1 AND NOT XCZ1 AND (X10Z1 OR X8Z1) THEN
						bRunOut := FALSE;
						SeqNo := 0;
				END_IF;
	20 : (* Clear HPR Request *)
				Result := FROM( TRUE, i_Start_IO_No, 817 + AxisOff, 1, wTmp);
				IF (wTmp AND H0008) <> 0 THEN
						Result := TO( TRUE, 1, i_Start_IO_No, 1521 + AxisOff, 1);
				END_IF;
				SeqNo := 21;
	21 : (* Wait *)
				Result := FROM( TRUE, i_Start_IO_No, 1521 + AxisOff, 1, wTmp);
				IF wTmp = 0 THEN
						SeqNo := 0;
				END_IF;
END_CASE;
 	
b_Run := bRunOut;
END_FUNCTION_BLOCK
